FUNCTION ClearData : BOOL
VAR_INPUT
	data : ANY;
END_VAR

MEMSET(destAddr := data.pValue, fillByte := 0, n := TO_UDINT(data.diSize));

END_FUNCTION

(* stored: Version 1.1.0.1, ProductVersion 3.1.4024.12
   POU ClearData: Id {8eb72f59-ecbe-098c-3744-6112c41f7ebc}, SpecialFunc None *)
